RoboDK station: RoboDK_VersionFinal.rdk

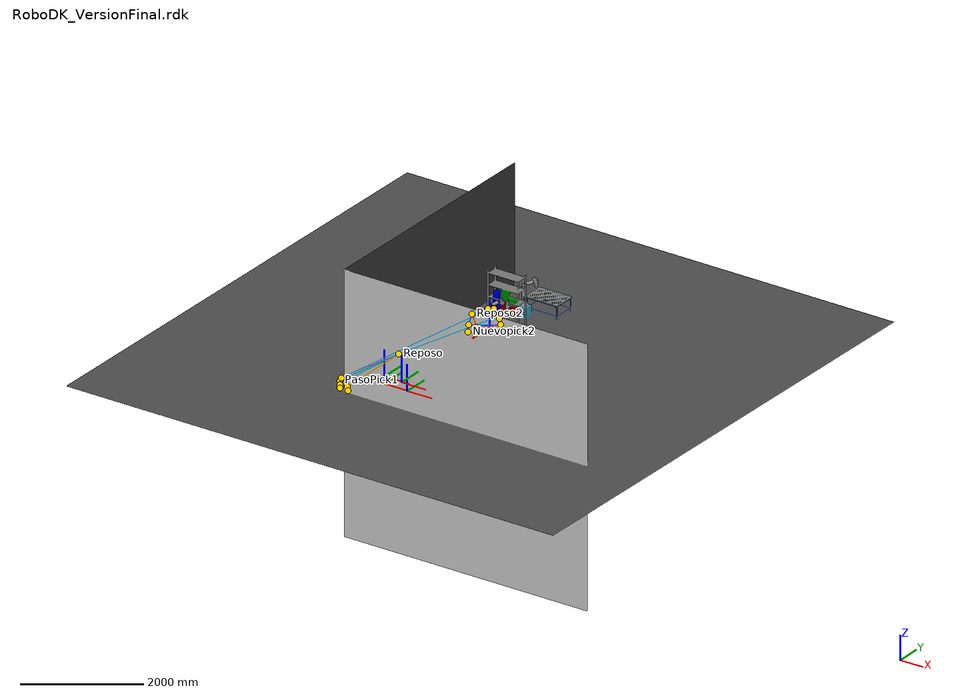
[picture v0: the station drawn from its stored meshes, robots at their saved joint values, targets as dots, program paths as lines]
Station RoboDK_VersionFinal (saved by RoboDK 5.9.4). Poses are relative to the parent item; angles as X-Y-Z fixed-axis rotations.
Station parameters (name, value as stored): IO_5, 1, pedido_id, 3, pedido_tipo, enantyum, pedido_posicion, X01-Y03, pedido_resultado, ok
  - frame UR3e Base - Clasificación at (400, 3450, 0) mm, rotated rx 0 ry 0 rz -90 deg
    - robot UR3e - Clasificaci (model UR3e): 6 axes, payload 3 kg, reach 500 mm, repeatability 0.03 mm, weight 11 kg
        modified DH rows (alpha deg, a mm, theta deg, d mm): 0, 0, 0, 151.9; 90, 0, 180, 0; 0, 243.55, 0, 0; 0, 213.2, 0, 131.05; -90, 0, 0, 85.35; 90, 0, 180, 92.1
        joint limits [-360, -360, -360, -360, -360, -360] to [360, 360, 360, 360, 360, 360]; home [0, -90, -90, 0, 90, 0]; saved at [130.788, -87.81, -66.397, -108.453, 84.697, 21.441]
      - tool RobotiQ EPick Vacuum Gripper (1 Cup), TCP at (0, 0, 130) mm, size 75 x 83 x 136.1 mm
    - target Reposo2 (Cartesian target) at (424.11, -46.06, 399.9) mm, rotated rx -137.59 ry 6.02 rz -87.52 deg; joints [13.28, -91.48, -57.54, -78.3, 87.11, 12.01] of UR3e - Clasificaci
    - object base - clasificaci at (0, 0, -100) mm, rotated rx 90 ry 0 rz 0 deg, size 170 x 200 x 170 mm, geometry from olaquease.obj
  - frame UR3e Base - Despaletizado at (50, 1000, 0) mm
    - robot UR3e - Despaletizado (model UR3e): 6 axes, payload 3 kg, reach 500 mm, repeatability 0.03 mm, weight 11 kg
        modified DH rows (alpha deg, a mm, theta deg, d mm): 0, 0, 0, 151.9; 90, 0, 180, 0; 0, 243.55, 0, 0; 0, 213.2, 0, 131.05; -90, 0, 0, 85.35; 90, 0, 180, 92.1
        joint limits [-360, -360, -360, -360, -360, -360] to [360, 360, 360, 360, 360, 360]; home [0, -90, -90, 0, 90, 0]; saved at [15.698, -84.751, -31.553, -98.733, 77.366, 5.023]
      - tool OnRobot VGP20 Vacuum Gripper, TCP at (-36, 0, 106.49) mm, size 268.4 x 184.1 x 103.7 mm
    - target Reposo (Cartesian target) at (336.1, -92.12, 531.02) mm, rotated rx -124.13 ry -3.06 rz -87.54 deg; joints [0.63, -91.59, -31.74, -90.74, 89.8, -3.56] of UR3e - Despaletizado
    - object base - despaletizado at (0, 0, -100) mm, rotated rx 90 ry 0 rz 0 deg, size 170 x 200 x 170 mm, geometry from olaquease.obj
  - frame cinta - despaletizado at (200, 775, 0) mm
    - robot cinta: 1 axes
        modified DH rows (alpha deg, a mm, theta deg, d mm): 0, 0, 0, 0 linear
        base shift (0, 0, 0) mm, rotated rx 0 ry 90 rz 0 deg
        joint limits [425] to [2000]; home [0]; saved at [450]
      - frame Frame 10 at (0, 0, 0) mm
        - frame Frame_Caja at (-250, 200, 0) mm
          - target Pick1 (Cartesian target) at (139.89, -13.23, 94.59) mm, rotated rx -179.32 ry 0 rz -90.91 deg; joints [11.689, -127.545, -60.36, -81.431, 89.852, 12.598] of UR3e - Despaletizado
          - target Pick2 (Cartesian target) at (-5.95, -20.92, 97.87) mm, rotated rx -179.32 ry 0 rz -90.91 deg; joints [15.948, -91.701, -109.286, -68.363, 89.803, 16.857] of UR3e - Despaletizado
          - target PasoPick (Cartesian target) at (-6.64, 14.1, 202.86) mm, rotated rx -179.32 ry 0 rz -90.91 deg; joints [15.815, -88.174, -90.444, -90.732, 89.804, 16.724] of UR3e - Despaletizado
          - target PasoPick1 (Cartesian target) at (-6.72, -20.9, 162.87) mm, rotated rx -179.32 ry 0 rz -90.91 deg; joints [15.992, -88.247, -94.806, -86.296, 89.802, 16.901] of UR3e - Despaletizado
          - target Pick1-abajo (Cartesian target) at (140.66, -13.24, 29.59) mm, rotated rx -179.32 ry 0 rz -90.91 deg; joints [11.667, -132.164, -70.38, -66.792, 89.852, 12.576] of UR3e - Despaletizado
          - target Pick2-abajo (Cartesian target) at (-5.24, -20.93, 37.87) mm, rotated rx -179.32 ry 0 rz -90.91 deg; joints [15.908, -99.569, -119.052, -50.728, 89.803, 16.817] of UR3e - Despaletizado
        - frame Frame_Caja at (-250, 200, 0) mm
          - target Pick1 (Cartesian target) at (139.89, -13.23, 94.59) mm, rotated rx -179.32 ry 0 rz -90.91 deg; joints [11.689, -127.545, -60.36, -81.431, 89.852, 12.598] of UR3e - Despaletizado
          - target Pick2 (Cartesian target) at (-5.95, -20.92, 97.87) mm, rotated rx -179.32 ry 0 rz -90.91 deg; joints [15.948, -91.701, -109.286, -68.363, 89.803, 16.857] of UR3e - Despaletizado
          - target PasoPick (Cartesian target) at (-6.64, 14.1, 202.86) mm, rotated rx -179.32 ry 0 rz -90.91 deg; joints [15.815, -88.174, -90.444, -90.732, 89.804, 16.724] of UR3e - Despaletizado
          - target PasoPick1 (Cartesian target) at (-6.72, -20.9, 162.87) mm, rotated rx -179.32 ry 0 rz -90.91 deg; joints [15.992, -88.247, -94.806, -86.296, 89.802, 16.901] of UR3e - Despaletizado
          - target Pick1-abajo (Cartesian target) at (140.66, -13.24, 29.59) mm, rotated rx -179.32 ry 0 rz -90.91 deg; joints [11.667, -132.164, -70.38, -66.792, 89.852, 12.576] of UR3e - Despaletizado
          - target Pick2-abajo (Cartesian target) at (-5.24, -20.93, 37.87) mm, rotated rx -179.32 ry 0 rz -90.91 deg; joints [15.908, -99.569, -119.052, -50.728, 89.803, 16.817] of UR3e - Despaletizado
        - frame Frame_Caja at (-250, 200, 0) mm
          - target Pick1 (Cartesian target) at (139.89, -13.23, 94.59) mm, rotated rx -179.32 ry 0 rz -90.91 deg; joints [11.689, -127.545, -60.36, -81.431, 89.852, 12.598] of UR3e - Despaletizado
          - target Pick2 (Cartesian target) at (-5.95, -20.92, 97.87) mm, rotated rx -179.32 ry 0 rz -90.91 deg; joints [15.948, -91.701, -109.286, -68.363, 89.803, 16.857] of UR3e - Despaletizado
          - target PasoPick (Cartesian target) at (-6.64, 14.1, 202.86) mm, rotated rx -179.32 ry 0 rz -90.91 deg; joints [15.815, -88.174, -90.444, -90.732, 89.804, 16.724] of UR3e - Despaletizado
          - target PasoPick1 (Cartesian target) at (-6.72, -20.9, 162.87) mm, rotated rx -179.32 ry 0 rz -90.91 deg; joints [15.992, -88.247, -94.806, -86.296, 89.802, 16.901] of UR3e - Despaletizado
          - target Pick1-abajo (Cartesian target) at (140.66, -13.24, 29.59) mm, rotated rx -179.32 ry 0 rz -90.91 deg; joints [11.667, -132.164, -70.38, -66.792, 89.852, 12.576] of UR3e - Despaletizado
          - target Pick2-abajo (Cartesian target) at (-5.24, -20.93, 37.87) mm, rotated rx -179.32 ry 0 rz -90.91 deg; joints [15.908, -99.569, -119.052, -50.728, 89.803, 16.817] of UR3e - Despaletizado
        - frame Frame_Caja at (-250, 200, 0) mm
          - target Pick1 (Cartesian target) at (139.89, -13.23, 94.59) mm, rotated rx -179.32 ry 0 rz -90.91 deg; joints [11.689, -127.545, -60.36, -81.431, 89.852, 12.598] of UR3e - Despaletizado
          - target Pick2 (Cartesian target) at (-5.95, -20.92, 97.87) mm, rotated rx -179.32 ry 0 rz -90.91 deg; joints [15.948, -91.701, -109.286, -68.363, 89.803, 16.857] of UR3e - Despaletizado
          - target PasoPick (Cartesian target) at (-6.64, 14.1, 202.86) mm, rotated rx -179.32 ry 0 rz -90.91 deg; joints [15.815, -88.174, -90.444, -90.732, 89.804, 16.724] of UR3e - Despaletizado
          - target PasoPick1 (Cartesian target) at (-6.72, -20.9, 162.87) mm, rotated rx -179.32 ry 0 rz -90.91 deg; joints [15.992, -88.247, -94.806, -86.296, 89.802, 16.901] of UR3e - Despaletizado
          - target Pick1-abajo (Cartesian target) at (140.66, -13.24, 29.59) mm, rotated rx -179.32 ry 0 rz -90.91 deg; joints [11.667, -132.164, -70.38, -66.792, 89.852, 12.576] of UR3e - Despaletizado
          - target Pick2-abajo (Cartesian target) at (-5.24, -20.93, 37.87) mm, rotated rx -179.32 ry 0 rz -90.91 deg; joints [15.908, -99.569, -119.052, -50.728, 89.803, 16.817] of UR3e - Despaletizado
        - frame Frame_Caja at (-250, 200, 0) mm
          - target Pick1 (Cartesian target) at (139.89, -13.23, 94.59) mm, rotated rx -179.32 ry 0 rz -90.91 deg; joints [11.689, -127.545, -60.36, -81.431, 89.852, 12.598] of UR3e - Despaletizado
          - target Pick2 (Cartesian target) at (-5.95, -20.92, 97.87) mm, rotated rx -179.32 ry 0 rz -90.91 deg; joints [15.948, -91.701, -109.286, -68.363, 89.803, 16.857] of UR3e - Despaletizado
          - target PasoPick (Cartesian target) at (-6.64, 14.1, 202.86) mm, rotated rx -179.32 ry 0 rz -90.91 deg; joints [15.815, -88.174, -90.444, -90.732, 89.804, 16.724] of UR3e - Despaletizado
          - target PasoPick1 (Cartesian target) at (-6.72, -20.9, 162.87) mm, rotated rx -179.32 ry 0 rz -90.91 deg; joints [15.992, -88.247, -94.806, -86.296, 89.802, 16.901] of UR3e - Despaletizado
          - target Pick1-abajo (Cartesian target) at (140.66, -13.24, 29.59) mm, rotated rx -179.32 ry 0 rz -90.91 deg; joints [11.667, -132.164, -70.38, -66.792, 89.852, 12.576] of UR3e - Despaletizado
          - target Pick2-abajo (Cartesian target) at (-5.24, -20.93, 37.87) mm, rotated rx -179.32 ry 0 rz -90.91 deg; joints [15.908, -99.569, -119.052, -50.728, 89.803, 16.817] of UR3e - Despaletizado
        - frame Frame_Caja at (-250, 200, 0) mm
          - target Pick1 (Cartesian target) at (139.89, -13.23, 94.59) mm, rotated rx -179.32 ry 0 rz -90.91 deg; joints [11.689, -127.545, -60.36, -81.431, 89.852, 12.598] of UR3e - Despaletizado
          - target Pick2 (Cartesian target) at (-5.95, -20.92, 97.87) mm, rotated rx -179.32 ry 0 rz -90.91 deg; joints [15.948, -91.701, -109.286, -68.363, 89.803, 16.857] of UR3e - Despaletizado
          - target PasoPick (Cartesian target) at (-6.64, 14.1, 202.86) mm, rotated rx -179.32 ry 0 rz -90.91 deg; joints [15.815, -88.174, -90.444, -90.732, 89.804, 16.724] of UR3e - Despaletizado
          - target PasoPick1 (Cartesian target) at (-6.72, -20.9, 162.87) mm, rotated rx -179.32 ry 0 rz -90.91 deg; joints [15.992, -88.247, -94.806, -86.296, 89.802, 16.901] of UR3e - Despaletizado
          - target Pick1-abajo (Cartesian target) at (140.66, -13.24, 29.59) mm, rotated rx -179.32 ry 0 rz -90.91 deg; joints [11.667, -132.164, -70.38, -66.792, 89.852, 12.576] of UR3e - Despaletizado
          - target Pick2-abajo (Cartesian target) at (-5.24, -20.93, 37.87) mm, rotated rx -179.32 ry 0 rz -90.91 deg; joints [15.908, -99.569, -119.052, -50.728, 89.803, 16.817] of UR3e - Despaletizado
        - frame Frame_Caja at (-250, 200, 0) mm
          - target Pick1 (Cartesian target) at (139.89, -13.23, 94.59) mm, rotated rx -179.32 ry 0 rz -90.91 deg; joints [11.689, -127.545, -60.36, -81.431, 89.852, 12.598] of UR3e - Despaletizado
          - target Pick2 (Cartesian target) at (-5.95, -20.92, 97.87) mm, rotated rx -179.32 ry 0 rz -90.91 deg; joints [15.948, -91.701, -109.286, -68.363, 89.803, 16.857] of UR3e - Despaletizado
          - target PasoPick (Cartesian target) at (-6.64, 14.1, 202.86) mm, rotated rx -179.32 ry 0 rz -90.91 deg; joints [15.815, -88.174, -90.444, -90.732, 89.804, 16.724] of UR3e - Despaletizado
          - target PasoPick1 (Cartesian target) at (-6.72, -20.9, 162.87) mm, rotated rx -179.32 ry 0 rz -90.91 deg; joints [15.992, -88.247, -94.806, -86.296, 89.802, 16.901] of UR3e - Despaletizado
          - target Pick1-abajo (Cartesian target) at (140.66, -13.24, 29.59) mm, rotated rx -179.32 ry 0 rz -90.91 deg; joints [11.667, -132.164, -70.38, -66.792, 89.852, 12.576] of UR3e - Despaletizado
          - target Pick2-abajo (Cartesian target) at (-5.24, -20.93, 37.87) mm, rotated rx -179.32 ry 0 rz -90.91 deg; joints [15.908, -99.569, -119.052, -50.728, 89.803, 16.817] of UR3e - Despaletizado
        - frame Frame_Caja at (-250, 200, 0) mm
          - target Pick1 (Cartesian target) at (139.89, -13.23, 94.59) mm, rotated rx -179.32 ry 0 rz -90.91 deg; joints [11.689, -127.545, -60.36, -81.431, 89.852, 12.598] of UR3e - Despaletizado
          - target Pick2 (Cartesian target) at (-5.95, -20.92, 97.87) mm, rotated rx -179.32 ry 0 rz -90.91 deg; joints [15.948, -91.701, -109.286, -68.363, 89.803, 16.857] of UR3e - Despaletizado
          - target PasoPick (Cartesian target) at (-6.64, 14.1, 202.86) mm, rotated rx -179.32 ry 0 rz -90.91 deg; joints [15.815, -88.174, -90.444, -90.732, 89.804, 16.724] of UR3e - Despaletizado
          - target PasoPick1 (Cartesian target) at (-6.72, -20.9, 162.87) mm, rotated rx -179.32 ry 0 rz -90.91 deg; joints [15.992, -88.247, -94.806, -86.296, 89.802, 16.901] of UR3e - Despaletizado
          - target Pick1-abajo (Cartesian target) at (140.66, -13.24, 29.59) mm, rotated rx -179.32 ry 0 rz -90.91 deg; joints [11.667, -132.164, -70.38, -66.792, 89.852, 12.576] of UR3e - Despaletizado
          - target Pick2-abajo (Cartesian target) at (-5.24, -20.93, 37.87) mm, rotated rx -179.32 ry 0 rz -90.91 deg; joints [15.908, -99.569, -119.052, -50.728, 89.803, 16.817] of UR3e - Despaletizado
        - frame Frame_Caja at (-250, 200, 0) mm
          - target Pick1 (Cartesian target) at (139.89, -13.23, 94.59) mm, rotated rx -179.32 ry 0 rz -90.91 deg; joints [11.689, -127.545, -60.36, -81.431, 89.852, 12.598] of UR3e - Despaletizado
          - target Pick2 (Cartesian target) at (-5.95, -20.92, 97.87) mm, rotated rx -179.32 ry 0 rz -90.91 deg; joints [15.948, -91.701, -109.286, -68.363, 89.803, 16.857] of UR3e - Despaletizado
          - target PasoPick (Cartesian target) at (-6.64, 14.1, 202.86) mm, rotated rx -179.32 ry 0 rz -90.91 deg; joints [15.815, -88.174, -90.444, -90.732, 89.804, 16.724] of UR3e - Despaletizado
          - target PasoPick1 (Cartesian target) at (-6.72, -20.9, 162.87) mm, rotated rx -179.32 ry 0 rz -90.91 deg; joints [15.992, -88.247, -94.806, -86.296, 89.802, 16.901] of UR3e - Despaletizado
          - target Pick1-abajo (Cartesian target) at (140.66, -13.24, 29.59) mm, rotated rx -179.32 ry 0 rz -90.91 deg; joints [11.667, -132.164, -70.38, -66.792, 89.852, 12.576] of UR3e - Despaletizado
          - target Pick2-abajo (Cartesian target) at (-5.24, -20.93, 37.87) mm, rotated rx -179.32 ry 0 rz -90.91 deg; joints [15.908, -99.569, -119.052, -50.728, 89.803, 16.817] of UR3e - Despaletizado
        - frame Frame_Caja at (-250, 200, 0) mm
          - target Pick1 (Cartesian target) at (139.89, -13.23, 94.59) mm, rotated rx -179.32 ry 0 rz -90.91 deg; joints [11.689, -127.545, -60.36, -81.431, 89.852, 12.598] of UR3e - Despaletizado
          - target Pick2 (Cartesian target) at (-5.95, -20.92, 97.87) mm, rotated rx -179.32 ry 0 rz -90.91 deg; joints [15.948, -91.701, -109.286, -68.363, 89.803, 16.857] of UR3e - Despaletizado
          - target PasoPick (Cartesian target) at (-6.64, 14.1, 202.86) mm, rotated rx -179.32 ry 0 rz -90.91 deg; joints [15.815, -88.174, -90.444, -90.732, 89.804, 16.724] of UR3e - Despaletizado
          - target PasoPick1 (Cartesian target) at (-6.72, -20.9, 162.87) mm, rotated rx -179.32 ry 0 rz -90.91 deg; joints [15.992, -88.247, -94.806, -86.296, 89.802, 16.901] of UR3e - Despaletizado
          - target Pick1-abajo (Cartesian target) at (140.66, -13.24, 29.59) mm, rotated rx -179.32 ry 0 rz -90.91 deg; joints [11.667, -132.164, -70.38, -66.792, 89.852, 12.576] of UR3e - Despaletizado
          - target Pick2-abajo (Cartesian target) at (-5.24, -20.93, 37.87) mm, rotated rx -179.32 ry 0 rz -90.91 deg; joints [15.908, -99.569, -119.052, -50.728, 89.803, 16.817] of UR3e - Despaletizado
        - frame Frame_Caja at (-250, 200, 0) mm
          - target Pick1 (Cartesian target) at (139.89, -13.23, 94.59) mm, rotated rx -179.32 ry 0 rz -90.91 deg; joints [11.689, -127.545, -60.36, -81.431, 89.852, 12.598] of UR3e - Despaletizado
          - target Pick2 (Cartesian target) at (-5.95, -20.92, 97.87) mm, rotated rx -179.32 ry 0 rz -90.91 deg; joints [15.948, -91.701, -109.286, -68.363, 89.803, 16.857] of UR3e - Despaletizado
          - target PasoPick (Cartesian target) at (-6.64, 14.1, 202.86) mm, rotated rx -179.32 ry 0 rz -90.91 deg; joints [15.815, -88.174, -90.444, -90.732, 89.804, 16.724] of UR3e - Despaletizado
          - target PasoPick1 (Cartesian target) at (-6.72, -20.9, 162.87) mm, rotated rx -179.32 ry 0 rz -90.91 deg; joints [15.992, -88.247, -94.806, -86.296, 89.802, 16.901] of UR3e - Despaletizado
          - target Pick1-abajo (Cartesian target) at (140.66, -13.24, 29.59) mm, rotated rx -179.32 ry 0 rz -90.91 deg; joints [11.667, -132.164, -70.38, -66.792, 89.852, 12.576] of UR3e - Despaletizado
          - target Pick2-abajo (Cartesian target) at (-5.24, -20.93, 37.87) mm, rotated rx -179.32 ry 0 rz -90.91 deg; joints [15.908, -99.569, -119.052, -50.728, 89.803, 16.817] of UR3e - Despaletizado
        - frame Frame_Caja at (-250, 200, 0) mm
          - target Pick1 (Cartesian target) at (139.89, -13.23, 94.59) mm, rotated rx -179.32 ry 0 rz -90.91 deg; joints [11.689, -127.545, -60.36, -81.431, 89.852, 12.598] of UR3e - Despaletizado
          - target Pick2 (Cartesian target) at (-5.95, -20.92, 97.87) mm, rotated rx -179.32 ry 0 rz -90.91 deg; joints [15.948, -91.701, -109.286, -68.363, 89.803, 16.857] of UR3e - Despaletizado
          - target PasoPick (Cartesian target) at (-6.64, 14.1, 202.86) mm, rotated rx -179.32 ry 0 rz -90.91 deg; joints [15.815, -88.174, -90.444, -90.732, 89.804, 16.724] of UR3e - Despaletizado
          - target PasoPick1 (Cartesian target) at (-6.72, -20.9, 162.87) mm, rotated rx -179.32 ry 0 rz -90.91 deg; joints [15.992, -88.247, -94.806, -86.296, 89.802, 16.901] of UR3e - Despaletizado
          - target Pick1-abajo (Cartesian target) at (140.66, -13.24, 29.59) mm, rotated rx -179.32 ry 0 rz -90.91 deg; joints [11.667, -132.164, -70.38, -66.792, 89.852, 12.576] of UR3e - Despaletizado
          - target Pick2-abajo (Cartesian target) at (-5.24, -20.93, 37.87) mm, rotated rx -179.32 ry 0 rz -90.91 deg; joints [15.908, -99.569, -119.052, -50.728, 89.803, 16.817] of UR3e - Despaletizado
        - frame Frame_Caja at (-250, 200, 0) mm
          - target Pick1 (Cartesian target) at (139.89, -13.23, 94.59) mm, rotated rx -179.32 ry 0 rz -90.91 deg; joints [11.689, -127.545, -60.36, -81.431, 89.852, 12.598] of UR3e - Despaletizado
          - target Pick2 (Cartesian target) at (-5.95, -20.92, 97.87) mm, rotated rx -179.32 ry 0 rz -90.91 deg; joints [15.948, -91.701, -109.286, -68.363, 89.803, 16.857] of UR3e - Despaletizado
          - target PasoPick (Cartesian target) at (-6.64, 14.1, 202.86) mm, rotated rx -179.32 ry 0 rz -90.91 deg; joints [15.815, -88.174, -90.444, -90.732, 89.804, 16.724] of UR3e - Despaletizado
          - target PasoPick1 (Cartesian target) at (-6.72, -20.9, 162.87) mm, rotated rx -179.32 ry 0 rz -90.91 deg; joints [15.992, -88.247, -94.806, -86.296, 89.802, 16.901] of UR3e - Despaletizado
          - target Pick1-abajo (Cartesian target) at (140.66, -13.24, 29.59) mm, rotated rx -179.32 ry 0 rz -90.91 deg; joints [11.667, -132.164, -70.38, -66.792, 89.852, 12.576] of UR3e - Despaletizado
          - target Pick2-abajo (Cartesian target) at (-5.24, -20.93, 37.87) mm, rotated rx -179.32 ry 0 rz -90.91 deg; joints [15.908, -99.569, -119.052, -50.728, 89.803, 16.817] of UR3e - Despaletizado
        - frame Frame_Caja at (-250, 200, 0) mm
          - target Pick1 (Cartesian target) at (139.89, -13.23, 94.59) mm, rotated rx -179.32 ry 0 rz -90.91 deg; joints [11.689, -127.545, -60.36, -81.431, 89.852, 12.598] of UR3e - Despaletizado
          - target Pick2 (Cartesian target) at (-5.95, -20.92, 97.87) mm, rotated rx -179.32 ry 0 rz -90.91 deg; joints [15.948, -91.701, -109.286, -68.363, 89.803, 16.857] of UR3e - Despaletizado
          - target PasoPick (Cartesian target) at (-6.64, 14.1, 202.86) mm, rotated rx -179.32 ry 0 rz -90.91 deg; joints [15.815, -88.174, -90.444, -90.732, 89.804, 16.724] of UR3e - Despaletizado
          - target PasoPick1 (Cartesian target) at (-6.72, -20.9, 162.87) mm, rotated rx -179.32 ry 0 rz -90.91 deg; joints [15.992, -88.247, -94.806, -86.296, 89.802, 16.901] of UR3e - Despaletizado
          - target Pick1-abajo (Cartesian target) at (140.66, -13.24, 29.59) mm, rotated rx -179.32 ry 0 rz -90.91 deg; joints [11.667, -132.164, -70.38, -66.792, 89.852, 12.576] of UR3e - Despaletizado
          - target Pick2-abajo (Cartesian target) at (-5.24, -20.93, 37.87) mm, rotated rx -179.32 ry 0 rz -90.91 deg; joints [15.908, -99.569, -119.052, -50.728, 89.803, 16.817] of UR3e - Despaletizado
        - frame Frame_Caja at (-250, 200, 0) mm
          - target Pick1 (Cartesian target) at (139.89, -13.23, 94.59) mm, rotated rx -179.32 ry 0 rz -90.91 deg; joints [11.689, -127.545, -60.36, -81.431, 89.852, 12.598] of UR3e - Despaletizado
          - target Pick2 (Cartesian target) at (-5.95, -20.92, 97.87) mm, rotated rx -179.32 ry 0 rz -90.91 deg; joints [15.948, -91.701, -109.286, -68.363, 89.803, 16.857] of UR3e - Despaletizado
          - target PasoPick (Cartesian target) at (-6.64, 14.1, 202.86) mm, rotated rx -179.32 ry 0 rz -90.91 deg; joints [15.815, -88.174, -90.444, -90.732, 89.804, 16.724] of UR3e - Despaletizado
          - target PasoPick1 (Cartesian target) at (-6.72, -20.9, 162.87) mm, rotated rx -179.32 ry 0 rz -90.91 deg; joints [15.992, -88.247, -94.806, -86.296, 89.802, 16.901] of UR3e - Despaletizado
          - target Pick1-abajo (Cartesian target) at (140.66, -13.24, 29.59) mm, rotated rx -179.32 ry 0 rz -90.91 deg; joints [11.667, -132.164, -70.38, -66.792, 89.852, 12.576] of UR3e - Despaletizado
          - target Pick2-abajo (Cartesian target) at (-5.24, -20.93, 37.87) mm, rotated rx -179.32 ry 0 rz -90.91 deg; joints [15.908, -99.569, -119.052, -50.728, 89.803, 16.817] of UR3e - Despaletizado
        - frame Frame_Caja at (-250, 200, 0) mm
          - target Pick1 (Cartesian target) at (139.89, -13.23, 94.59) mm, rotated rx -179.32 ry 0 rz -90.91 deg; joints [11.689, -127.545, -60.36, -81.431, 89.852, 12.598] of UR3e - Despaletizado
          - target Pick2 (Cartesian target) at (-5.95, -20.92, 97.87) mm, rotated rx -179.32 ry 0 rz -90.91 deg; joints [15.948, -91.701, -109.286, -68.363, 89.803, 16.857] of UR3e - Despaletizado
          - target PasoPick (Cartesian target) at (-6.64, 14.1, 202.86) mm, rotated rx -179.32 ry 0 rz -90.91 deg; joints [15.815, -88.174, -90.444, -90.732, 89.804, 16.724] of UR3e - Despaletizado
          - target PasoPick1 (Cartesian target) at (-6.72, -20.9, 162.87) mm, rotated rx -179.32 ry 0 rz -90.91 deg; joints [15.992, -88.247, -94.806, -86.296, 89.802, 16.901] of UR3e - Despaletizado
          - target Pick1-abajo (Cartesian target) at (140.66, -13.24, 29.59) mm, rotated rx -179.32 ry 0 rz -90.91 deg; joints [11.667, -132.164, -70.38, -66.792, 89.852, 12.576] of UR3e - Despaletizado
          - target Pick2-abajo (Cartesian target) at (-5.24, -20.93, 37.87) mm, rotated rx -179.32 ry 0 rz -90.91 deg; joints [15.908, -99.569, -119.052, -50.728, 89.803, 16.817] of UR3e - Despaletizado
        - frame Frame_Caja at (-250, 200, 0) mm
          - target Pick1 (Cartesian target) at (139.89, -13.23, 94.59) mm, rotated rx -179.32 ry 0 rz -90.91 deg; joints [11.689, -127.545, -60.36, -81.431, 89.852, 12.598] of UR3e - Despaletizado
          - target Pick2 (Cartesian target) at (-5.95, -20.92, 97.87) mm, rotated rx -179.32 ry 0 rz -90.91 deg; joints [15.948, -91.701, -109.286, -68.363, 89.803, 16.857] of UR3e - Despaletizado
          - target PasoPick (Cartesian target) at (-6.64, 14.1, 202.86) mm, rotated rx -179.32 ry 0 rz -90.91 deg; joints [15.815, -88.174, -90.444, -90.732, 89.804, 16.724] of UR3e - Despaletizado
          - target PasoPick1 (Cartesian target) at (-6.72, -20.9, 162.87) mm, rotated rx -179.32 ry 0 rz -90.91 deg; joints [15.992, -88.247, -94.806, -86.296, 89.802, 16.901] of UR3e - Despaletizado
          - target Pick1-abajo (Cartesian target) at (140.66, -13.24, 29.59) mm, rotated rx -179.32 ry 0 rz -90.91 deg; joints [11.667, -132.164, -70.38, -66.792, 89.852, 12.576] of UR3e - Despaletizado
          - target Pick2-abajo (Cartesian target) at (-5.24, -20.93, 37.87) mm, rotated rx -179.32 ry 0 rz -90.91 deg; joints [15.908, -99.569, -119.052, -50.728, 89.803, 16.817] of UR3e - Despaletizado
        - frame Frame_Caja at (-250, 200, 0) mm
          - target Pick1 (Cartesian target) at (139.89, -13.23, 94.59) mm, rotated rx -179.32 ry 0 rz -90.91 deg; joints [11.689, -127.545, -60.36, -81.431, 89.852, 12.598] of UR3e - Despaletizado
          - target Pick2 (Cartesian target) at (-5.95, -20.92, 97.87) mm, rotated rx -179.32 ry 0 rz -90.91 deg; joints [15.948, -91.701, -109.286, -68.363, 89.803, 16.857] of UR3e - Despaletizado
          - target PasoPick (Cartesian target) at (-6.64, 14.1, 202.86) mm, rotated rx -179.32 ry 0 rz -90.91 deg; joints [15.815, -88.174, -90.444, -90.732, 89.804, 16.724] of UR3e - Despaletizado
          - target PasoPick1 (Cartesian target) at (-6.72, -20.9, 162.87) mm, rotated rx -179.32 ry 0 rz -90.91 deg; joints [15.992, -88.247, -94.806, -86.296, 89.802, 16.901] of UR3e - Despaletizado
          - target Pick1-abajo (Cartesian target) at (140.66, -13.24, 29.59) mm, rotated rx -179.32 ry 0 rz -90.91 deg; joints [11.667, -132.164, -70.38, -66.792, 89.852, 12.576] of UR3e - Despaletizado
          - target Pick2-abajo (Cartesian target) at (-5.24, -20.93, 37.87) mm, rotated rx -179.32 ry 0 rz -90.91 deg; joints [15.908, -99.569, -119.052, -50.728, 89.803, 16.817] of UR3e - Despaletizado
        - frame Frame_Caja at (-250, 200, 0) mm
          - target Pick1 (Cartesian target) at (139.89, -13.23, 94.59) mm, rotated rx -179.32 ry 0 rz -90.91 deg; joints [11.689, -127.545, -60.36, -81.431, 89.852, 12.598] of UR3e - Despaletizado
          - target Pick2 (Cartesian target) at (-5.95, -20.92, 97.87) mm, rotated rx -179.32 ry 0 rz -90.91 deg; joints [15.948, -91.701, -109.286, -68.363, 89.803, 16.857] of UR3e - Despaletizado
          - target PasoPick (Cartesian target) at (-6.64, 14.1, 202.86) mm, rotated rx -179.32 ry 0 rz -90.91 deg; joints [15.815, -88.174, -90.444, -90.732, 89.804, 16.724] of UR3e - Despaletizado
          - target PasoPick1 (Cartesian target) at (-6.72, -20.9, 162.87) mm, rotated rx -179.32 ry 0 rz -90.91 deg; joints [15.992, -88.247, -94.806, -86.296, 89.802, 16.901] of UR3e - Despaletizado
          - target Pick1-abajo (Cartesian target) at (140.66, -13.24, 29.59) mm, rotated rx -179.32 ry 0 rz -90.91 deg; joints [11.667, -132.164, -70.38, -66.792, 89.852, 12.576] of UR3e - Despaletizado
          - target Pick2-abajo (Cartesian target) at (-5.24, -20.93, 37.87) mm, rotated rx -179.32 ry 0 rz -90.91 deg; joints [15.908, -99.569, -119.052, -50.728, 89.803, 16.817] of UR3e - Despaletizado
        - frame Frame_Caja at (-250, 200, 0) mm
          - target Pick1 (Cartesian target) at (139.89, -13.23, 94.59) mm, rotated rx -179.32 ry 0 rz -90.91 deg; joints [11.689, -127.545, -60.36, -81.431, 89.852, 12.598] of UR3e - Despaletizado
          - target Pick2 (Cartesian target) at (-5.95, -20.92, 97.87) mm, rotated rx -179.32 ry 0 rz -90.91 deg; joints [15.948, -91.701, -109.286, -68.363, 89.803, 16.857] of UR3e - Despaletizado
          - target PasoPick (Cartesian target) at (-6.64, 14.1, 202.86) mm, rotated rx -179.32 ry 0 rz -90.91 deg; joints [15.815, -88.174, -90.444, -90.732, 89.804, 16.724] of UR3e - Despaletizado
          - target PasoPick1 (Cartesian target) at (-6.72, -20.9, 162.87) mm, rotated rx -179.32 ry 0 rz -90.91 deg; joints [15.992, -88.247, -94.806, -86.296, 89.802, 16.901] of UR3e - Despaletizado
          - target Pick1-abajo (Cartesian target) at (140.66, -13.24, 29.59) mm, rotated rx -179.32 ry 0 rz -90.91 deg; joints [11.667, -132.164, -70.38, -66.792, 89.852, 12.576] of UR3e - Despaletizado
          - target Pick2-abajo (Cartesian target) at (-5.24, -20.93, 37.87) mm, rotated rx -179.32 ry 0 rz -90.91 deg; joints [15.908, -99.569, -119.052, -50.728, 89.803, 16.817] of UR3e - Despaletizado
        - frame Frame_Caja at (-250, 200, 0) mm
          - target Pick1 (Cartesian target) at (139.89, -13.23, 94.59) mm, rotated rx -179.32 ry 0 rz -90.91 deg; joints [11.689, -127.545, -60.36, -81.431, 89.852, 12.598] of UR3e - Despaletizado
          - target Pick2 (Cartesian target) at (-5.95, -20.92, 97.87) mm, rotated rx -179.32 ry 0 rz -90.91 deg; joints [15.948, -91.701, -109.286, -68.363, 89.803, 16.857] of UR3e - Despaletizado
          - target PasoPick (Cartesian target) at (-6.64, 14.1, 202.86) mm, rotated rx -179.32 ry 0 rz -90.91 deg; joints [15.815, -88.174, -90.444, -90.732, 89.804, 16.724] of UR3e - Despaletizado
          - target PasoPick1 (Cartesian target) at (-6.72, -20.9, 162.87) mm, rotated rx -179.32 ry 0 rz -90.91 deg; joints [15.992, -88.247, -94.806, -86.296, 89.802, 16.901] of UR3e - Despaletizado
          - target Pick1-abajo (Cartesian target) at (140.66, -13.24, 29.59) mm, rotated rx -179.32 ry 0 rz -90.91 deg; joints [11.667, -132.164, -70.38, -66.792, 89.852, 12.576] of UR3e - Despaletizado
          - target Pick2-abajo (Cartesian target) at (-5.24, -20.93, 37.87) mm, rotated rx -179.32 ry 0 rz -90.91 deg; joints [15.908, -99.569, -119.052, -50.728, 89.803, 16.817] of UR3e - Despaletizado
        - frame Frame_Caja at (-250, 200, 0) mm
          - target Pick1 (Cartesian target) at (139.89, -13.23, 94.59) mm, rotated rx -179.32 ry 0 rz -90.91 deg; joints [11.689, -127.545, -60.36, -81.431, 89.852, 12.598] of UR3e - Despaletizado
          - target Pick2 (Cartesian target) at (-5.95, -20.92, 97.87) mm, rotated rx -179.32 ry 0 rz -90.91 deg; joints [15.948, -91.701, -109.286, -68.363, 89.803, 16.857] of UR3e - Despaletizado
          - target PasoPick (Cartesian target) at (-6.64, 14.1, 202.86) mm, rotated rx -179.32 ry 0 rz -90.91 deg; joints [15.815, -88.174, -90.444, -90.732, 89.804, 16.724] of UR3e - Despaletizado
          - target PasoPick1 (Cartesian target) at (-6.72, -20.9, 162.87) mm, rotated rx -179.32 ry 0 rz -90.91 deg; joints [15.992, -88.247, -94.806, -86.296, 89.802, 16.901] of UR3e - Despaletizado
          - target Pick1-abajo (Cartesian target) at (140.66, -13.24, 29.59) mm, rotated rx -179.32 ry 0 rz -90.91 deg; joints [11.667, -132.164, -70.38, -66.792, 89.852, 12.576] of UR3e - Despaletizado
          - target Pick2-abajo (Cartesian target) at (-5.24, -20.93, 37.87) mm, rotated rx -179.32 ry 0 rz -90.91 deg; joints [15.908, -99.569, -119.052, -50.728, 89.803, 16.817] of UR3e - Despaletizado
    - object pata1 at (50, 20, -200) mm, size 50 x 50 x 150 mm, geometry from Cylinder-50x150mm.sld
    - object pata2 at (50, 410, -200) mm, size 50 x 50 x 150 mm, geometry from Cylinder-50x150mm.sld
    - object pata3 at (2000, 25, -200) mm, size 50 x 50 x 150 mm, geometry from Cylinder-50x150mm.sld
    - object pata4 at (2000, 410, -190) mm, size 50 x 50 x 150 mm, geometry from Cylinder-50x150mm.sld
  - frame cinta - clasificación at (175, 3250, 0) mm, rotated rx 0 ry 0 rz -90 deg
    - robot cinta 2: 1 axes
        modified DH rows (alpha deg, a mm, theta deg, d mm): 0, 0, 0, 0 linear
        base shift (0, 0, 0) mm, rotated rx 0 ry 90 rz 0 deg
        joint limits [-400] to [2000]; home [0]; saved at [-400]
      - frame Frame_despaletizadas at (0, 5050, 0) mm
        - frame Frame_place_desp1 at (0, 150, 0) mm
          - target Paso1 (Cartesian target) at (-13.08, -5145.35, 202.9) mm, rotated rx -179.31 ry 0 rz 56.73 deg; joints [80.175, -87.842, -84.404, -97.123, 89.724, 23.445] of UR3e - Despaletizado
          - target Paso2 (Cartesian target) at (-60.46, -5061.67, 204.51) mm, rotated rx -178.44 ry -3.78 rz 86.72 deg; joints [70.316, -108.237, -61.222, -97.975, 86.819, -16.522] of UR3e - Despaletizado
          - target Place Despaletizado (Cartesian target) at (-95.9, -4983.44, 30.92) mm, rotated rx -178.44 ry 1.22 rz 86.85 deg; joints [60.153, -137.173, -60.813, -71.172, 91.79, -26.668] of UR3e - Despaletizado
          - target PrePlace_despaletizado (Cartesian target) at (-94.48, -4982.44, 81.11) mm, rotated rx -178.44 ry 1.22 rz 86.85 deg; joints [59.961, -134.066, -52.685, -82.412, 91.793, -26.861] of UR3e - Despaletizado
        - frame Frame_place_desp2 at (220, 150, 0) mm
          - target Paso1 (Cartesian target) at (-13.08, -5145.35, 202.9) mm, rotated rx -179.31 ry 0 rz 56.73 deg; joints [80.175, -87.842, -84.404, -97.123, 89.724, 23.445] of UR3e - Despaletizado
          - target Paso2 (Cartesian target) at (-60.46, -5061.67, 204.51) mm, rotated rx -178.44 ry -3.78 rz 86.72 deg; joints [70.316, -108.237, -61.222, -97.975, 86.819, -16.522] of UR3e - Despaletizado
          - target Place Despaletizado (Cartesian target) at (-95.9, -4983.44, 30.92) mm, rotated rx -178.44 ry 1.22 rz 86.85 deg; joints [60.153, -137.173, -60.813, -71.172, 91.79, -26.668] of UR3e - Despaletizado
          - target PrePlace_despaletizado (Cartesian target) at (-94.48, -4982.44, 81.11) mm, rotated rx -178.44 ry 1.22 rz 86.85 deg; joints [59.961, -134.066, -52.685, -82.412, 91.793, -26.861] of UR3e - Despaletizado
        - frame Frame_place_desp3 at (450, 150, 0) mm
          - target Paso1 (Cartesian target) at (-13.08, -5145.35, 202.9) mm, rotated rx -179.31 ry 0 rz 56.73 deg; joints [80.175, -87.842, -84.404, -97.123, 89.724, 23.445] of UR3e - Despaletizado
          - target Paso2 (Cartesian target) at (-60.46, -5061.67, 204.51) mm, rotated rx -178.44 ry -3.78 rz 86.72 deg; joints [70.316, -108.237, -61.222, -97.975, 86.819, -16.522] of UR3e - Despaletizado
          - target Place Despaletizado (Cartesian target) at (-95.9, -4983.44, 30.92) mm, rotated rx -178.44 ry 1.22 rz 86.85 deg; joints [60.153, -137.173, -60.813, -71.172, 91.79, -26.668] of UR3e - Despaletizado
          - target PrePlace_despaletizado (Cartesian target) at (-94.48, -4982.44, 81.11) mm, rotated rx -178.44 ry 1.22 rz 86.85 deg; joints [59.961, -134.066, -52.685, -82.412, 91.793, -26.861] of UR3e - Despaletizado
        - frame Frame_place_desp4 at (650, 150, 0) mm
          - target Paso1 (Cartesian target) at (-13.08, -5145.35, 202.9) mm, rotated rx -179.31 ry 0 rz 56.73 deg; joints [80.175, -87.842, -84.404, -97.123, 89.724, 23.445] of UR3e - Despaletizado
          - target Paso2 (Cartesian target) at (-60.46, -5061.67, 204.51) mm, rotated rx -178.44 ry -3.78 rz 86.72 deg; joints [70.316, -108.237, -61.222, -97.975, 86.819, -16.522] of UR3e - Despaletizado
          - target Place Despaletizado (Cartesian target) at (-95.9, -4983.44, 30.92) mm, rotated rx -178.44 ry 1.22 rz 86.85 deg; joints [60.153, -137.173, -60.813, -71.172, 91.79, -26.668] of UR3e - Despaletizado
          - target PrePlace_despaletizado (Cartesian target) at (-94.48, -4982.44, 81.11) mm, rotated rx -178.44 ry 1.22 rz 86.85 deg; joints [59.961, -134.066, -52.685, -82.412, 91.793, -26.861] of UR3e - Despaletizado
    - object pata1 - 2 at (50, 20, -200) mm, rotated rx 0 ry 0 rz 90 deg, size 50 x 50 x 150 mm, geometry from Cylinder-50x150mm.sld
    - object pata2 - 2 at (50, 410, -200) mm, size 50 x 50 x 150 mm, geometry from Cylinder-50x150mm.sld
    - object pata3 - 2 at (2000, 25, -200) mm, size 50 x 50 x 150 mm, geometry from Cylinder-50x150mm.sld
    - object pata4 - 2 at (2000, 410, -190) mm, size 50 x 50 x 150 mm, geometry from Cylinder-50x150mm.sld
    - frame Frame Pick Clasificacion at (0, 5200, 0) mm
      - target PrePick_clasif2 (Cartesian target) at (232.44, -5084.56, 187.8) mm, rotated rx -179.98 ry -2.95 rz -81.23 deg; joints [4.402, -122.109, -44.04, -103.606, 87.063, -4.376] of UR3e - Clasificaci
      - target Pick_clasif2 (Cartesian target) at (233.47, -5090.86, 62.97) mm, rotated rx -179.46 ry -2.89 rz -91.48 deg; joints [3.54, -124.29, -74.53, -70.89, 87.07, 5] of UR3e - Clasificaci
      - target Pick_clasif1 (Cartesian target) at (232.87, -4940.49, 61.49) mm, rotated rx -179.31 ry -2.87 rz -91.32 deg; joints [23.68, -121.62, -79.01, -69.96, 87.11, 25] of UR3e - Clasificaci
      - target PrePick_clasif1 (Cartesian target) at (231.51, -4934.23, 186.29) mm, rotated rx -179.99 ry -2.95 rz -78.08 deg; joints [24.552, -118.971, -49.099, -102.568, 87.119, 12.649] of UR3e - Clasificaci
      - target Paso (Cartesian target) at (39.67, -4578.8, 252) mm, rotated rx -168.07 ry -0.24 rz -26.24 deg; joints [76.72, -118.97, -36.89, -102.56, 87.11, 12.64] of UR3e - Clasificaci
      - target Paso2 (Cartesian target) at (-348.42, -4656.59, 306.9) mm, rotated rx -173.21 ry -2.13 rz 42.51 deg; joints [138.85, -99.16, -44.86, -119.46, 87.15, 6.05] of UR3e - Clasificaci
      - target Paso4 (Cartesian target) at (-233.56, -4760.65, 389.01) mm, rotated rx -142.29 ry 2.04 rz 42.48 deg; joints [140, -49.13, -75.05, -108.16, 87.01, 7.2] of UR3e - Clasificaci
      - object infrared sensor - proximity sensor (1) at (190, -5250, 0) mm, rotated rx 0 ry 0 rz 90 deg, size 100 x 42.7 x 42.7 mm, geometry from infrared sensor - proximity sensor (1).stl
      - target Nuevopick1 (Cartesian target) at (239.54, -4940.77, 61.55) mm, rotated rx -179.39 ry -1.29 rz -92.71 deg; joints [22.499, -123.163, -76.629, -70.206, 88.576, 25.201] of UR3e - Clasificaci
      - target Nuevopick2 (Cartesian target) at (233.61, -5087.33, 62.84) mm, rotated rx -179.41 ry -1.33 rz -92.4 deg; joints [3.204, -124.422, -74.353, -70.766, 88.621, 5.588] of UR3e - Clasificaci
  - frame Sistema - Estantería at (400, 4050, -173.38) mm
    - target Place 1 (Cartesian target) at (-22.93, -204.87, 525.14) mm, rotated rx -90 ry 0 rz 0 deg; joints [207.93, -116.903, -92.388, 29.291, 62.07, 0] of UR3e - Clasificaci
    - target Target 2 (Cartesian target) at (322.8, -521.68, 452.98) mm, rotated rx -171.23 ry -2.21 rz -71.16 deg; joints [130.788, -87.631, -67.051, -107.978, 84.697, 21.441] of UR3e - Clasificaci
    - target Place_base (Cartesian target) at (-213.83, -204.87, 379.68) mm, rotated rx -90 ry 0 rz 0 deg; joints [259.472, -135.813, -115.812, 71.625, 10.528, 0] of UR3e - Clasificaci
    - object Estanteria at (0, 0, 0) mm, size 624.2 x 963.2 x 234 mm, geometry from eb_metal_shelf_01.obj
    - target Target 3 (Cartesian target) at (400.79, -632.87, 393.4) mm, rotated rx -168.07 ry -0.24 rz -116.24 deg; joints [109.466, -99.497, -72.038, -90.245, 81.324, 45.055] of UR3e - Clasificaci
    - target Pick_base_antes (Cartesian target) at (-213.89, -129.51, 378.2) mm, rotated rx -89.91 ry 1.64 rz 177.07 deg; joints [-103.271, -145.254, -88.344, 53.694, 100.334, 1.652] of UR3e - pedidos
    - target Paso_ped3 (Cartesian target) at (-131.82, 121.32, 662.13) mm, rotated rx -90.23 ry 1.63 rz -178.38 deg; joints [-98.637, -52.41, -111.868, -15.952, 100.265, 1.587] of UR3e - pedidos
    - target Paso_ped4 (Cartesian target) at (-126.77, 42.59, 563.07) mm, rotated rx -90.23 ry 1.63 rz -178.38 deg; joints [-91.201, -64.707, -134.036, 18.516, 92.829, 1.617] of UR3e - pedidos
    - target Paso_ped5 (Cartesian target) at (-214.08, 164.54, 606.19) mm, rotated rx -90.23 ry 1.63 rz -178.38 deg; joints [-135.362, -83.287, -109.019, 11.974, 136.989, 1.385] of UR3e - pedidos
    - target Paso_ped6 (Cartesian target) at (-291.93, 214.82, 509.51) mm, rotated rx -90.23 ry 1.63 rz -178.38 deg; joints [-161.185, -113.423, -102.583, 35.24, 162.811, 0.896] of UR3e - pedidos
    - target Pick_base (Cartesian target) at (-192.17, -40.89, 371.84) mm, rotated rx -88.66 ry 1.64 rz 177.07 deg; joints [18.618, -41.504, 115.771, 102.085, 338.369, -354.973] of UR3e - pedidos
    - object Prism 9-2 at (-148.31, -139.79, 308.56) mm, rotated rx 17.47 ry 88.43 rz -72.45 deg, size 62.5 x 125 x 62.5 mm, geometry from Prism-250x125x125mm.sld
    - object Prism 10-2 at (-0.05, -141.61, 308.76) mm, rotated rx 6.04 ry 88.51 rz -83.84 deg, size 62.5 x 125 x 62.5 mm, geometry from Prism-250x125x125mm.sld
    - object Prism 7-2 at (164.42, -138.64, 308.62) mm, rotated rx 17.47 ry 88.43 rz -72.45 deg, size 62.5 x 125 x 62.5 mm, geometry from Prism-250x125x125mm.sld
    - object Prism 8-2 at (-152.32, -140.45, 523.8) mm, rotated rx 6.04 ry 88.51 rz -83.84 deg, size 62.5 x 125 x 62.5 mm, geometry from Prism-250x125x125mm.sld
    - object Prism 5-2 at (12.15, -137.48, 523.67) mm, rotated rx 17.47 ry 88.43 rz -72.45 deg, size 62.5 x 125 x 62.5 mm, geometry from Prism-250x125x125mm.sld
    - object Prism 6-2 at (160.41, -139.29, 523.84) mm, rotated rx 6.04 ry 88.51 rz -83.84 deg, size 62.5 x 125 x 62.5 mm, geometry from Prism-250x125x125mm.sld
    - object Prism 3-2 at (-137.85, -135.49, 368.76) mm, rotated rx 17.47 ry 88.43 rz -72.45 deg, size 62.5 x 125 x 62.5 mm, geometry from Prism-250x125x125mm.sld
    - object Prism 4-2 at (10.37, -137.3, 368.89) mm, rotated rx 6.04 ry 88.51 rz -83.84 deg, size 62.5 x 125 x 62.5 mm, geometry from Prism-250x125x125mm.sld
    - object Prism 1-2 at (174.88, -134.33, 368.81) mm, rotated rx 17.47 ry 88.43 rz -72.45 deg, size 62.5 x 125 x 62.5 mm, geometry from Prism-250x125x125mm.sld
    - object Prism 2-2 at (-141.9, -136.14, 583.93) mm, rotated rx 6.04 ry 88.51 rz -83.84 deg, size 62.5 x 125 x 62.5 mm, geometry from Prism-250x125x125mm.sld
    - object Prism 9 at (7.18, -144.86, 580.48) mm, rotated rx 17.47 ry 88.43 rz -72.45 deg, size 62.5 x 125 x 62.5 mm, geometry from Prism-250x125x125mm.sld
    - object Prism 7 at (-145.09, -143.7, 431.53) mm, rotated rx 17.47 ry 88.43 rz -72.45 deg, size 62.5 x 125 x 62.5 mm, geometry from Prism-250x125x125mm.sld
    - object Prism 8 at (3.12, -145.52, 431.71) mm, rotated rx 6.04 ry 88.51 rz -83.84 deg, size 62.5 x 125 x 62.5 mm, geometry from Prism-250x125x125mm.sld
    - object Prism 3 at (17.16, -135.47, 643.47) mm, rotated rx 17.47 ry 88.43 rz -72.45 deg, size 62.5 x 125 x 62.5 mm, geometry from Prism-250x125x125mm.sld
  - frame Frame 6 at (-250, 200, 0) mm
    - object tinker at (0, 0, -10) mm, size 400 x 300 x 125 mm, geometry from tinker.obj
    - target Pick1 (Cartesian target) at (139.89, -13.23, 94.59) mm, rotated rx -179.32 ry 0 rz -90.91 deg; joints [11.689, -127.545, -60.36, -81.431, 89.852, 12.598] of UR3e - Despaletizado
    - target Pick2 (Cartesian target) at (-5.95, -20.92, 97.87) mm, rotated rx -179.32 ry 0 rz -90.91 deg; joints [15.948, -91.701, -109.286, -68.363, 89.803, 16.857] of UR3e - Despaletizado
    - target PasoPick (Cartesian target) at (-6.64, 14.1, 202.86) mm, rotated rx -179.32 ry 0 rz -90.91 deg; joints [15.815, -88.174, -90.444, -90.732, 89.804, 16.724] of UR3e - Despaletizado
    - target PasoPick1 (Cartesian target) at (-6.72, -20.9, 162.87) mm, rotated rx -179.32 ry 0 rz -90.91 deg; joints [15.992, -88.247, -94.806, -86.296, 89.802, 16.901] of UR3e - Despaletizado
    - target Pick1-abajo (Cartesian target) at (140.66, -13.24, 29.59) mm, rotated rx -179.32 ry 0 rz -90.91 deg; joints [11.667, -132.164, -70.38, -66.792, 89.852, 12.576] of UR3e - Despaletizado
    - target Pick2-abajo (Cartesian target) at (-5.24, -20.93, 37.87) mm, rotated rx -179.32 ry 0 rz -90.91 deg; joints [15.908, -99.569, -119.052, -50.728, 89.803, 16.817] of UR3e - Despaletizado
    - object Prism 2-2 at (-80, 90, 60) mm, size 62.5 x 125 x 62.5 mm, geometry from Prism-250x125x125mm.sld
    - object Prism 1-2 at (-80, -50, 60) mm, size 62.5 x 125 x 62.5 mm, geometry from Prism-250x125x125mm.sld
    - object Prism 4-2 at (-10, 90, 60) mm, size 62.5 x 125 x 62.5 mm, geometry from Prism-250x125x125mm.sld
    - object Prism 3-2 at (-10, -50, 60) mm, size 62.5 x 125 x 62.5 mm, geometry from Prism-250x125x125mm.sld
    - object Prism 5-2 at (60, -50, 60) mm, size 62.5 x 125 x 62.5 mm, geometry from Prism-250x125x125mm.sld
    - object Prism 6-2 at (60, 90, 60) mm, size 62.5 x 125 x 62.5 mm, geometry from Prism-250x125x125mm.sld
    - object Prism 9-2 at (200, -50, 60) mm, size 62.5 x 125 x 62.5 mm, geometry from Prism-250x125x125mm.sld
    - object Prism 10-2 at (200, 90, 60) mm, size 62.5 x 125 x 62.5 mm, geometry from Prism-250x125x125mm.sld
    - object Prism 7-2 at (130, -50, 60) mm, size 62.5 x 125 x 62.5 mm, geometry from Prism-250x125x125mm.sld
    - object Prism 8-2 at (130, 90, 60) mm, size 62.5 x 125 x 62.5 mm, geometry from Prism-250x125x125mm.sld
    - object Prism 2 at (-80, 90, 0) mm, size 62.5 x 125 x 62.5 mm, geometry from Prism-250x125x125mm.sld
    - object Prism 250x125x125mm at (-80, -50, 0) mm, size 62.5 x 125 x 62.5 mm, geometry from Prism-250x125x125mm.sld
    - object Prism 4 at (-10, 90, 0) mm, size 62.5 x 125 x 62.5 mm, geometry from Prism-250x125x125mm.sld
    - object Prism 3 at (-10, -50, 0) mm, size 62.5 x 125 x 62.5 mm, geometry from Prism-250x125x125mm.sld
    - object Prism 5 at (60, -50, 0) mm, size 62.5 x 125 x 62.5 mm, geometry from Prism-250x125x125mm.sld
    - object Prism 6 at (60, 90, 0) mm, size 62.5 x 125 x 62.5 mm, geometry from Prism-250x125x125mm.sld
    - object Prism 9 at (200, -50, 0) mm, size 62.5 x 125 x 62.5 mm, geometry from Prism-250x125x125mm.sld
    - object Prism 10 at (200, 90, 0) mm, size 62.5 x 125 x 62.5 mm, geometry from Prism-250x125x125mm.sld
    - object Prism 7 at (130, -50, 0) mm, size 62.5 x 125 x 62.5 mm, geometry from Prism-250x125x125mm.sld
    - object Prism 8 at (130, 90, 0) mm, size 62.5 x 125 x 62.5 mm, geometry from Prism-250x125x125mm.sld
  - frame Frame_sensor at (-50, 500, 0) mm
    - object infrared sensor - proximity sensor (1) at (300, 200, 0) mm, rotated rx 0 ry 0 rz 90 deg, size 100 x 42.7 x 42.7 mm, geometry from infrared sensor - proximity sensor (1).stl
  - frame UR3e Base - pedidos at (400, 4430, 0) mm
    - robot UR3e - pedidos (model UR3e): 6 axes, payload 3 kg, reach 500 mm, repeatability 0.03 mm, weight 11 kg
        modified DH rows (alpha deg, a mm, theta deg, d mm): 0, 0, 0, 151.9; 90, 0, 180, 0; 0, 243.55, 0, 0; 0, 213.2, 0, 131.05; -90, 0, 0, 85.35; 90, 0, 180, 92.1
        joint limits [-360, -360, -360, -360, -360, -360] to [360, 360, 360, 360, 360, 360]; home [0, -90, -90, 0, 90, 0]; saved at [33.678, -87.094, -74.931, 0.727, 9.729, -13.917]
      - tool RobotiQ EPick Vacuum Gripper (1 Cup), TCP at (0, 0, 130) mm, size 75 x 83 x 136.1 mm
    - object base - pedidos at (0, 0, -100) mm, rotated rx 90 ry 0 rz 0 deg, size 170 x 200 x 170 mm, geometry from olaquease.obj
    - object Mesa_pedidos at (0, 400, 65) mm, size 636.3 x 422.1 x 252 mm, geometry from Table-2000x1200x800mm.sld
    - frame Frame_pedidos at (0, 400, 65) mm
      - target Place_pedido (Cartesian target) at (384.34, -165.38, 46.78) mm, rotated rx -90.39 ry 0.12 rz -1.35 deg; joints [22.113, -167.141, -69.546, 55.718, 156.539, -0.769] of UR3e - pedidos
      - target Pre_pedidos (Cartesian target) at (383.36, -207.27, 47.06) mm, rotated rx -90.39 ry 0.12 rz -1.35 deg; joints [15.783, -167.001, -69.826, 55.518, 162.867, -1.131] of UR3e - pedidos
      - target Paso_ped2 (Cartesian target) at (474.36, -412.99, 243.96) mm, rotated rx -84.74 ry -1.58 rz -64.81 deg; joints [4.98, -121.46, -105.569, 52.639, 110.266, 0.365] of UR3e - pedidos
      - target Paso_ped1 (Cartesian target) at (421, -495.79, 270.65) mm, rotated rx -84.67 ry 1.35 rz -95.59 deg; joints [17.594, -99.316, -130.185, 55.297, 66.796, -0.937] of UR3e - pedidos
      - target Reposo_pedidos (Cartesian target) at (359.35, -581.08, 488.81) mm, rotated rx -86.88 ry 4.53 rz -136.85 deg; joints [33.678, -87.094, -74.931, 0.727, 9.729, -13.917] of UR3e - pedidos
  - folder Clasificacion
    - program Pick2 (14 instructions, listed below)
    - program Pick1 (14 instructions, listed below)
  - folder Despaletizado
    - program PickPlace-Despaletizado1 (39 instructions, listed below)
    - program PickPlace-Despaletizado2 (33 instructions, listed below)
    - program PickPlace-Despaletizado3 (38 instructions, listed below)
    - program PickPlace-Despaletizado4 (34 instructions, listed below)
    - program Programa Despaletizado (22 instructions, listed below)
  - folder Python
    - Python program Reset (listed below)
    - Python program ApareceCaja (listed below)
    - Python program AvanzaCaja (listed below)
    - Python program CintaPick (listed below)
    - Python program AvanzaPlace (listed below)
    - Python program ResetPick (listed below)
    - Python program AvanzaPick (listed below)
    - Python program ProgramaClasificacion (listed below)
    - Python program Pedidos_PickPlace_base (listed below)
    - Python program Pedidos_PickPlace (listed below)
  - program ProgramaPrincipal (2 instructions, listed below)
  - object Square at (600, 2900, -200) mm, size 9600 x 9600 x 0 mm, geometry from Square.sld
    - object Square at (3800, 0, -200) mm, rotated rx 90 ry 0 rz 90 deg, size 4800 x 4800 x 0 mm, geometry from Square.sld
    - object Square at (-1000, 0, -200) mm, rotated rx 0 ry 90 rz 0 deg, size 4800 x 4800 x 0 mm, geometry from Square.sld
    - object Box 400x200mm (Closed) at (1200, -2200, 0) mm, rotated rx 90 ry 0 rz 90 deg, size 603.6 x 1201.8 x 650 mm, geometry from Box-400x200mm-Closed.sld
    - object Square at (1400, 2400, -200) mm, rotated rx 90 ry 0 rz 0 deg, size 4800 x 4800 x 0 mm, geometry from Square.sld
    - object Square at (1400, -2400, -200) mm, rotated rx 90 ry 0 rz 0 deg, size 4800 x 4800 x 0 mm, geometry from Square.sld
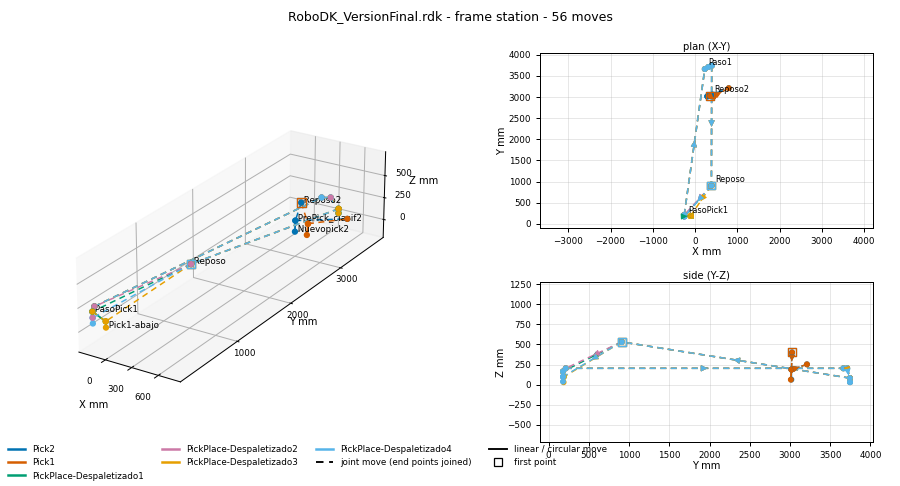
[picture p0: tool path of RoboDK_VersionFinal.rdk in frame station, 56 of 56 moves have a stored position in this frame; points joined in program order, loops and branches not executed]

--- program Pick2 (robot UR3e - Clasificaci) ---
  Est. Ref.: UR3e Base - Clasificación
  Establecer velocidad (500.0 mm/s)
  Est. herr: RobotiQ EPick Vacuum Gripper (1 Cup)
  MoveJ (Reposo2)
  Est. Ref.: Frame Pick Clasificacion
  MoveJ (PrePick_clasif2)
  Establecer velocidad (100.0 mm/s)
  MoveL (Nuevopick2)
  Set IO_5=1
  Adjuntar a RobotiQ EPick Vacuum Gripper (1 Cup)
  Pausa 2.0 s
  MoveL (PrePick_clasif2)
  Establecer velocidad (500.0 mm/s)
  MoveJ (Paso)

--- program Pick1 (robot UR3e - Clasificaci) ---
  Est. Ref.: UR3e Base - Clasificación
  Establecer velocidad (500.0 mm/s)
  Est. herr: RobotiQ EPick Vacuum Gripper (1 Cup)
  MoveJ (Reposo2)
  Est. Ref.: Frame Pick Clasificacion
  MoveJ (PrePick_clasif1)
  Establecer velocidad (100.0 mm/s)
  MoveL (Nuevopick1)
  Set IO_5=1
  Adjuntar a RobotiQ EPick Vacuum Gripper (1 Cup)
  Pausa 2.0 s
  MoveL (PrePick_clasif1)
  Establecer velocidad (500.0 mm/s)
  MoveJ (Paso)

--- program PickPlace-Despaletizado1 (robot UR3e - Despaletizado) ---
  Est. Ref.: UR3e Base - Despaletizado
  Establecer velocidad (500.0 mm/s)
  Est. herr: RobotiQ EPick Vacuum Gripper (1 Cup)
  MoveJ (Reposo)
  Est. Ref.: Frame_6_Copia at (350, -25, 0) mm
  MoveJ (PasoPick1)
  Establecer velocidad (100.0 mm/s)
  MoveL (Pick1)
  Set IO_5=1
  Adjuntar a OnRobot VGP20 Vacuum Gripper
  Adjuntar a OnRobot VGP20 Vacuum Gripper
  Adjuntar a OnRobot VGP20 Vacuum Gripper
  Adjuntar a OnRobot VGP20 Vacuum Gripper
  Adjuntar a OnRobot VGP20 Vacuum Gripper
  Adjuntar a OnRobot VGP20 Vacuum Gripper
  Pausa 2.0 s
  MoveL (PasoPick1)
  Establecer velocidad (500.0 mm/s)
  MoveJ (PasoPick)
  Est. Ref.: Frame_place_desp -> Frame_place_desp1
  MoveJ (Paso1)
  MoveJ (Paso2)
  MoveJ (PrePlace_despaletizado)
  Establecer velocidad (100.0 mm/s)
  MoveL (Place Despaletizado)
  Set IO_5=0
  Est. Ref.: Frame_despaletizadas
  Separar de OnRobot VGP20 Vacuum Gripper
  Separar de OnRobot VGP20 Vacuum Gripper
  Separar de OnRobot VGP20 Vacuum Gripper
  Separar de OnRobot VGP20 Vacuum Gripper
  Separar de OnRobot VGP20 Vacuum Gripper
  Separar de OnRobot VGP20 Vacuum Gripper
  Pausa 2.0 s
  Est. Ref.: Frame_place_desp -> Frame_place_desp1
  MoveL (PrePlace_despaletizado)
  Establecer velocidad (500.0 mm/s)
  Est. Ref.: UR3e Base - Despaletizado
  MoveJ (Reposo)

--- program PickPlace-Despaletizado2 (robot UR3e - Despaletizado) ---
  Est. Ref.: UR3e Base - Despaletizado
  Establecer velocidad (500.0 mm/s)
  Est. herr: RobotiQ EPick Vacuum Gripper (1 Cup)
  MoveJ (Reposo)
  Est. Ref.: Frame_6_Copia at (350, -25, 0) mm
  MoveJ (PasoPick)
  Establecer velocidad (100.0 mm/s)
  MoveL (Pick2)
  Set IO_5=1
  Adjuntar a OnRobot VGP20 Vacuum Gripper
  Adjuntar a OnRobot VGP20 Vacuum Gripper
  Adjuntar a OnRobot VGP20 Vacuum Gripper
  Adjuntar a OnRobot VGP20 Vacuum Gripper
  Pausa 2.0 s
  MoveL (PasoPick1)
  Establecer velocidad (500.0 mm/s)
  MoveJ (PasoPick)
  Est. Ref.: Frame_place_desp2
  MoveJ (Paso1)
  MoveJ (Paso2)
  MoveJ (PrePlace_despaletizado)
  Establecer velocidad (100.0 mm/s)
  MoveL (Place Despaletizado)
  Set IO_5=0
  Separar de OnRobot VGP20 Vacuum Gripper
  Separar de OnRobot VGP20 Vacuum Gripper
  Separar de OnRobot VGP20 Vacuum Gripper
  Separar de OnRobot VGP20 Vacuum Gripper
  Pausa 2.0 s
  MoveL (PrePlace_despaletizado)
  Establecer velocidad (500.0 mm/s)
  Est. Ref.: UR3e Base - Despaletizado
  MoveJ (Reposo)

--- program PickPlace-Despaletizado3 (robot UR3e - Despaletizado) ---
  Est. Ref.: UR3e Base - Despaletizado
  Establecer velocidad (500.0 mm/s)
  Est. herr: RobotiQ EPick Vacuum Gripper (1 Cup)
  MoveJ (Reposo)
  Est. Ref.: Frame_6_Copia at (350, -25, 0) mm
  MoveJ (Pick1)
  Establecer velocidad (100.0 mm/s)
  MoveL (Pick1-abajo)
  Set IO_5=1
  Adjuntar a OnRobot VGP20 Vacuum Gripper
  Adjuntar a OnRobot VGP20 Vacuum Gripper
  Adjuntar a OnRobot VGP20 Vacuum Gripper
  Adjuntar a OnRobot VGP20 Vacuum Gripper
  Adjuntar a OnRobot VGP20 Vacuum Gripper
  Adjuntar a OnRobot VGP20 Vacuum Gripper
  Pausa 2.0 s
  MoveL (Pick1)
  Establecer velocidad (500.0 mm/s)
  MoveJ (PasoPick1)
  MoveJ (PasoPick)
  Est. Ref.: Frame_place_desp3
  MoveJ (Paso1)
  MoveJ (Paso2)
  MoveJ (PrePlace_despaletizado)
  Establecer velocidad (100.0 mm/s)
  MoveL (Place Despaletizado)
  Set IO_5=0
  Separar de OnRobot VGP20 Vacuum Gripper
  Separar de OnRobot VGP20 Vacuum Gripper
  Separar de OnRobot VGP20 Vacuum Gripper
  Separar de OnRobot VGP20 Vacuum Gripper
  Separar de OnRobot VGP20 Vacuum Gripper
  Separar de OnRobot VGP20 Vacuum Gripper
  Pausa 2.0 s
  MoveL (PrePlace_despaletizado)
  Establecer velocidad (500.0 mm/s)
  Est. Ref.: UR3e Base - Despaletizado
  MoveJ (Reposo)

--- program PickPlace-Despaletizado4 (robot UR3e - Despaletizado) ---
  Est. Ref.: UR3e Base - Despaletizado
  Establecer velocidad (500.0 mm/s)
  Est. herr: RobotiQ EPick Vacuum Gripper (1 Cup)
  MoveJ (Reposo)
  Est. Ref.: Frame_6_Copia at (350, -25, 0) mm
  MoveJ (Pick2)
  Establecer velocidad (100.0 mm/s)
  MoveL (Pick2-abajo)
  Set IO_5=1
  Adjuntar a OnRobot VGP20 Vacuum Gripper
  Adjuntar a OnRobot VGP20 Vacuum Gripper
  Adjuntar a OnRobot VGP20 Vacuum Gripper
  Adjuntar a OnRobot VGP20 Vacuum Gripper
  Pausa 2.0 s
  MoveL (Pick2)
  Establecer velocidad (500.0 mm/s)
  MoveJ (PasoPick1)
  MoveJ (PasoPick)
  Est. Ref.: Frame_place_desp4
  MoveJ (Paso1)
  MoveJ (Paso2)
  MoveJ (Place Despaletizado)
  Establecer velocidad (100.0 mm/s)
  MoveL (Place Despaletizado)
  Set IO_5=0
  Separar de OnRobot VGP20 Vacuum Gripper
  Separar de OnRobot VGP20 Vacuum Gripper
  Separar de OnRobot VGP20 Vacuum Gripper
  Pausa 2.0 s
  Separar de OnRobot VGP20 Vacuum Gripper
  MoveL (PrePlace_despaletizado)
  Establecer velocidad (500.0 mm/s)
  Est. Ref.: UR3e Base - Despaletizado
  MoveJ (Reposo)

--- program Programa Despaletizado (robot cinta) ---
  Llamar Reset
  Llamar ResetPick
  Llamar ApareceCaja
  Llamar AvanzaCaja
  Llamar PickPlace-Despaletizado1
  Llamar AvanzaPlace
  Llamar AvanzaPlace
  Llamar AvanzaPlace
  Llamar AvanzaPlace
  Llamar AvanzaPlace
  Llamar PickPlace-Despaletizado2
  Llamar AvanzaPlace
  Llamar AvanzaPlace
  Llamar AvanzaPlace
  Llamar AvanzaPlace
  Llamar PickPlace-Despaletizado3
  Llamar AvanzaPlace
  Llamar AvanzaPlace
  Llamar AvanzaPlace
  Llamar AvanzaPlace
  Llamar PickPlace-Despaletizado4
  Llamar CintaPick

--- Python program Reset ---
# Type help("robodk.robolink") or help("robodk.robomath") for more information
# Press F5 to run the script
# Documentation: https://robodk.com/doc/en/RoboDK-API.html
# Reference:     https://robodk.com/doc/en/PythonAPI/robodk.html
# Note: It is not required to keep a copy of this file, your Python script is saved with your RDK project

# You can also use the new version of the API:
from robodk import robolink    # RoboDK API
from robodk import robomath    # Robot toolbox
RDK = robolink.Robolink()

cinta = RDK.Item('cinta')

if cinta.Valid():
    cinta.setJoints([2000])

--- Python program ApareceCaja ---
# Type help("robodk.robolink") or help("robodk.robomath") for more information
# Press F5 to run the script
# Documentation: https://robodk.com/doc/en/RoboDK-API.html
# Reference:     https://robodk.com/doc/en/PythonAPI/robodk.html

from robodk import robolink    # RoboDK API
from robodk import robomath    # Robot toolbox

RDK = robolink.Robolink()

cinta = RDK.Item('cinta')
INCREMENTO_MM = -1550
caja_grande = RDK.Item('tinker')
caja_grande.setParam('Collisions', '0')


# Conjunto original (Frame con TODAS las cajitas + tinker)
caja = RDK.Item('Frame 6')
tinker = RDK.Item('Frame_6_Copia')

# Frame de la cinta
SR_Cinta = RDK.Item('Frame 10')

def hacer_visible_recursivo(item):

    # Si es un target -> ocultarlo
    if item.Type() == robolink.ITEM_TYPE_TARGET:
        item.setVisible(False)
    else:
        item.setVisible(True)

    # Recorrer hijos
    for hijo in item.Childs():
        hacer_visible_recursivo(hijo)

if cinta.Valid() and caja.Valid():
    # -------------------------------------------------
    # BORRAR COPIAS EXISTENTES EN "Sistema - Estantería"
    # -------------------------------------------------
    estanteria = RDK.Item('Sistema - Estantería')

    if estanteria.Valid():
        hijos = estanteria.Childs()  # copia de la lista
        for item in hijos:
            if item.Valid() and item.Name().startswith('Prism'):
                item.Delete()

    if tinker.Valid():
        tinker.Delete()

    #Copiar una caja
    caja.Copy()
    caja_copia = RDK.Paste()
    caja_copia.setName('Frame_Caja')

    # Colocar la copia en el inicio de la cinta
    caja_copia.setParent(SR_Cinta)
    caja_copia.setPose(caja.Pose())
    caja_copia.setVisible(True)

    hacer_visible_recursivo(caja_copia)

--- Python program AvanzaCaja ---
# Type help("robodk.robolink") or help("robodk.robomath") for more information
# Press F5 to run the script
# Documentation: https://robodk.com/doc/en/RoboDK-API.html
# Reference:     https://robodk.com/doc/en/PythonAPI/robodk.html
# Note: It is not required to keep a copy of this file, your Python script is saved with your RDK project

# You can also use the new version of the API:
from robodk import robolink    # RoboDK API
from robodk import robomath    # Robot toolbox
RDK = robolink.Robolink()

cinta = RDK.Item('cinta')
INCREMENTO_MM = -1550
caja_grande = RDK.Item('tinker')
caja_grande.setParam('Collisions', '0')


# Conjunto original (Frame con TODAS las cajitas + tinker)
caja = RDK.Item('Frame 6')
tinker = RDK.Item('Frame_6_Copia')

if cinta.Valid() and caja.Valid():

    # Avanzar Cinta
    cinta.setSpeed(1000)
    cinta.setAcceleration(100)

    joints = cinta.Joints()
    joints[0] += INCREMENTO_MM
    cinta.MoveJ(joints)

--- Python program CintaPick ---
# Type help("robodk.robolink") or help("robodk.robomath") for more information
# Press F5 to run the script
# Documentation: https://robodk.com/doc/en/RoboDK-API.html
# Reference:     https://robodk.com/doc/en/PythonAPI/robodk.html
# Note: It is not required to keep a copy of this file, your Python script is saved with your RDK project

# You can also use the new version of the API:
from robodk import robolink    # RoboDK API
from robodk import robomath    # Robot toolbox
RDK = robolink.Robolink()

cinta = RDK.Item('cinta 2')
INCREMENTO_MM = -960
#caja = RDK.Item('Frame 11')
SR_Cinta = RDK.Item('Frame_despaletizadas')

if cinta.Valid():
    cinta.setSpeed(500)
    cinta.setAcceleration(500)
    cinta.MoveJ(cinta.Joints() + INCREMENTO_MM)

--- Python program AvanzaPlace ---
# Type help("robodk.robolink") or help("robodk.robomath") for more information
# Press F5 to run the script
# Documentation: https://robodk.com/doc/en/RoboDK-API.html
# Reference:     https://robodk.com/doc/en/PythonAPI/robodk.html
# Note: It is not required to keep a copy of this file, your Python script is saved with your RDK project

# You can also use the new version of the API:
from robodk import robolink    # RoboDK API
from robodk import robomath    # Robot toolbox
RDK = robolink.Robolink()

cinta = RDK.Item('cinta 2')
INCREMENTO_MM = -50
#caja = RDK.Item('Frame 11')
SR_Cinta = RDK.Item('Frame 11')

if cinta.Valid():
    cinta.setSpeed(200)        # velocidad constante
    cinta.setAcceleration(50) # opcional, mm/s^2
    cinta.MoveJ(cinta.Joints() + INCREMENTO_MM)

--- Python program ResetPick ---
# Type help("robodk.robolink") or help("robodk.robomath") for more information
# Press F5 to run the script
# Documentation: https://robodk.com/doc/en/RoboDK-API.html
# Reference:     https://robodk.com/doc/en/PythonAPI/robodk.html
# Note: It is not required to keep a copy of this file, your Python script is saved with your RDK project

# You can also use the new version of the API:
from robodk import robolink    # RoboDK API
from robodk import robomath    # Robot toolbox
RDK = robolink.Robolink()

cinta = RDK.Item('cinta 2')

if cinta.Valid():
    cinta.setJoints([2000])

--- Python program AvanzaPick ---
# Type help("robodk.robolink") or help("robodk.robomath") for more information
# Press F5 to run the script
# Documentation: https://robodk.com/doc/en/RoboDK-API.html
# Reference:     https://robodk.com/doc/en/PythonAPI/robodk.html
# Note: It is not required to keep a copy of this file, your Python script is saved with your RDK project

# You can also use the new version of the API:
from robodk import robolink    # RoboDK API
from robodk import robomath    # Robot toolbox
RDK = robolink.Robolink()

cinta = RDK.Item('cinta 2')
INCREMENTO_MM = -70
#caja = RDK.Item('Frame 11')
SR_Cinta = RDK.Item('Frame 11')

if cinta.Valid():
    cinta.setSpeed(500)        # velocidad constante
    cinta.setAcceleration(500) # opcional, mm/s^2
    cinta.MoveJ(cinta.Joints() + INCREMENTO_MM)

--- Python program ProgramaClasificacion ---
from robodk import *
from robolink import *

RDK = Robolink()
robot = RDK.Item('UR3e Base - Clasificación', ITEM_TYPE_ROBOT)

tool = RDK.Item("RobotiQ EPick Vacuum Gripper (1 Cup)", ITEM_TYPE_TOOL)
frame_est = RDK.Item('Sistema - Estantería')

#base = RDK.Item('Estanteria')
#pose_base = base.Pose()


#pose_base = pose_base * transl(0, 0, 280)

#♥ TARGETS

target_Punto_Paso_1 = RDK.Item('Paso', robolink.ITEM_TYPE_TARGET)
target_Punto_Paso_2 = RDK.Item('Target 2', robolink.ITEM_TYPE_TARGET)
target_Punto_Paso_3 = RDK.Item('Target 3', robolink.ITEM_TYPE_TARGET)
#target_Pre_Place = RDK.Item('PrePlace', robolink.ITEM_TYPE_TARGET)


target_Place = RDK.Item('Place_base', robolink.ITEM_TYPE_TARGET)
pose_base = target_Place.Pose()


# Parámetros
ancho_caja = 125
fondo_caja = 66
alto_caja = 62.5

gap = 30

dx = ancho_caja + gap
dy = fondo_caja + gap
dz = 215

cols = 3
rows = 2
levels = 3

contador = 0
max_cajas = 18

robot.setPoseFrame(frame_est)
robot.setPoseTool(tool)

pose_target = pose_base

for k in range(levels):
    for i in range(rows):
        for j in range(cols):

            if contador >= max_cajas:
                break

            # PICK

            if contador % 2 == 0:
                RDK.RunProgram("Pick1", True)
            else:
                RDK.RunProgram("Pick2", True)
                if contador == 5:
                    RDK.RunProgram("AvanzaPlace", True)
                    RDK.RunProgram("AvanzaPlace", True)
                    RDK.RunProgram("AvanzaPlace", False)
                elif contador == 9:
                    RDK.RunProgram("AvanzaPlace", True)
                    RDK.RunProgram("AvanzaPlace", False)
                elif(contador == 15):
                    RDK.RunProgram("AvanzaPlace", True)
                    RDK.RunProgram("AvanzaPick", False)
                else:
                    RDK.RunProgram("AvanzaPick", False)

            #tool.AttachClosest()   # o caja.AttachTo(tool)

            # -------------------
            # CALCULAR PLACE
            # -------------------
            #offset = transl(
                #j*dx + ancho_caja/2,
                #i*dy + fondo_caja/2,
                #k*dz + alto_caja/2
            #)

            if contador <= 5:
                offset = transl(
                    j*dx + ancho_caja/2,
                    -i*dz + fondo_caja,
                    0
                )
            elif contador > 5 and contador <= 11 :
                offset = transl(
                    j*dx + ancho_caja/2,
                    -i*dz,
                    0
                )
            elif contador > 11 and contador <= 17:
                if contador == 16 or contador == 17:
                    offset = transl(
                        j*dx + ancho_caja/2,
                        -i*dz - fondo_caja + 7,
                        0
                    )
                else:
                    offset = transl(
                        j*dx + ancho_caja/2,
                        -i*dz - fondo_caja,
                        0
                    )
            else:
                offset = transl(
                    j*dx + ancho_caja/2,
                    -i*dz + fondo_caja,
                    0
                )


            pose_target = pose_base * offset

            robot.setPoseFrame(frame_est)
            robot.setPoseTool(tool)

            # -------------------
            # PLACE
            # -------------------
            robot.MoveJ(target_Punto_Paso_3)

            robot.MoveJ(target_Punto_Paso_2)
            robot.MoveJ(pose_target * robomath.transl([0,-50,0]))
            robot.setSpeed(100,20)
            pause(0.5)
            robot.MoveL(pose_target)

            objetos = tool.Childs()
            if len(objetos) > 0:
                caja = objetos[0]
                caja.setParentStatic(frame_est)

            tool.DetachAll()

            robot.MoveL(pose_target * robomath.transl([0,-50,0]))
            robot.setSpeed(1000,100)
            robot.MoveJ(target_Punto_Paso_2)

            # o mejor:
            # caja.AttachTo(frame_est)

            contador += 1

--- Python program Pedidos_PickPlace_base ---
from robodk import *
from robolink import *

RDK = Robolink()

robot = RDK.Item('UR3e - pedidos', ITEM_TYPE_ROBOT)
tool = robot.getLink(ITEM_TYPE_TOOL)
frame_est = RDK.Item('Sistema - Estantería')
frame_pedidos = RDK.Item('Frame_pedidos')

t_paso3 = RDK.Item('Paso_ped3', ITEM_TYPE_TARGET)
t_paso4 = RDK.Item('Paso_ped4', ITEM_TYPE_TARGET)
t_paso5 = RDK.Item('Paso_ped5', ITEM_TYPE_TARGET)
t_paso6 = RDK.Item('Paso_ped6', ITEM_TYPE_TARGET)

t_reposo  = RDK.Item('Reposo_pedidos', ITEM_TYPE_TARGET)
t_paso1   = RDK.Item('Paso_ped1', ITEM_TYPE_TARGET)
t_paso2   = RDK.Item('Paso_ped2', ITEM_TYPE_TARGET)
t_preplace = RDK.Item('Pre_pedidos', ITEM_TYPE_TARGET)
t_place = RDK.Item('Place_pedido', ITEM_TYPE_TARGET)

t_pick_ref = RDK.Item('Pick_base_antes', ITEM_TYPE_TARGET)
pose_ref = t_pick_ref.Pose()

robot.setPoseFrame(frame_est)
robot.setPoseTool(tool)

pose_base = RDK.Item('Place_base', ITEM_TYPE_TARGET).Pose()
pose_target = pose_base

# BASE DE DATOS

medicamentos = {
    "ibuprofeno": [],
    "paracetamol": [],
    "enantyum": []
}


# PARÁMETROS

ancho_caja = 125
fondo_caja = 66
alto_caja = 62.5
gap = 30
dx = ancho_caja + gap
dz = 215
cols = 3
rows = 2
levels = 3
contador = 0
max_cajas = 18

# GENERAR POSICIONES

for k in range(levels):
    for i in range(rows):
        for j in range(cols):
            if contador >= max_cajas:
                break

            if contador <= 5:
                offset = transl(j*dx + ancho_caja/2, -i*dz + fondo_caja, 0)
                if contador == 0 or contador == 3:
                    medicamentos["ibuprofeno"].append(pose_target * offset)
                elif contador <= 2:
                    medicamentos["paracetamol"].append(pose_target * offset)
                else:
                    medicamentos["enantyum"].append(pose_target * offset)

            elif contador <= 11:
                offset = transl(j*dx + ancho_caja/2, -i*dz, 0)
                if contador == 6 or contador == 9:
                    medicamentos["ibuprofeno"].append(pose_target * offset)
                elif contador <= 8:
                    medicamentos["paracetamol"].append(pose_target * offset)
                else:
                    medicamentos["enantyum"].append(pose_target * offset)

            elif contador <= 17:
                if contador == 16 or contador == 17:
                    offset = transl(j*dx + ancho_caja/2, -i*dz - fondo_caja + 7, 0)
                else:
                    offset = transl(j*dx + ancho_caja/2, -i*dz - fondo_caja, 0)
                if contador == 12 or contador == 15:
                    medicamentos["ibuprofeno"].append(pose_target * offset)
                elif contador <= 14:
                    medicamentos["paracetamol"].append(pose_target * offset)
                else:
                    medicamentos["enantyum"].append(pose_target * offset)

            contador += 1

# FUNCIÓN PEDIDO

def pedir_medicamento(tipo):
    if tipo not in medicamentos or not medicamentos[tipo]:
        print("Sin stock de", tipo)
        return

    pose_place_pos = medicamentos[tipo].pop()

    pose_place = Mat(pose_ref)
    pose_place[0,3] = pose_place_pos[0,3]
    pose_place[1,3] = pose_place_pos[1,3]
    pose_place[2,3] = pose_place_pos[2,3]

    pose_up = Mat(pose_place)
    pose_up[1,3] += 100
    pose_pick = Mat(pose_place)
    pose_pick[1,3] += 60

    robot.MoveJ(t_paso3)
    robot.MoveJ(t_paso4)
    robot.MoveJ(t_paso5)
    robot.MoveJ(t_paso6)

    robot.MoveJ(pose_up)
    robot.setSpeed(100, 20)
    pause(0.5)
    robot.MoveL(pose_pick)

    tool.AttachClosest()
    robot.MoveL(pose_up)
    robot.setSpeed(1000, 100)

    robot.MoveJ(t_paso6)
    robot.MoveJ(t_paso5)
    robot.MoveJ(t_paso4)
    robot.MoveJ(t_paso3)

    robot.setPoseFrame(frame_pedidos)

    # PLACE
    robot.MoveJ(t_reposo)
    robot.MoveJ(t_paso1)
    robot.MoveJ(t_paso2)

    robot.MoveJ(t_preplace)
    robot.setSpeed(100, 20)
    pause(0.5)
    robot.MoveL(t_place)

    tool.DetachAll()
    robot.MoveL(t_preplace)
    robot.setSpeed(1000, 100)

    robot.MoveJ(t_paso2)
    robot.MoveJ(t_paso1)
    robot.MoveJ(t_reposo)

#  EJECUTAR

pedir_medicamento("enantyum")

--- Python program Pedidos_PickPlace ---
from robodk import *
from robolink import *

RDK = Robolink()

robot = RDK.Item('UR3e - pedidos', ITEM_TYPE_ROBOT)
tool = robot.getLink(ITEM_TYPE_TOOL)
frame_est = RDK.Item('Sistema - Estantería')
frame_pedidos = RDK.Item('Frame_pedidos')

t_paso3 = RDK.Item('Paso_ped3', ITEM_TYPE_TARGET)
t_paso4 = RDK.Item('Paso_ped4', ITEM_TYPE_TARGET)
t_paso5 = RDK.Item('Paso_ped5', ITEM_TYPE_TARGET)
t_paso6 = RDK.Item('Paso_ped6', ITEM_TYPE_TARGET)

t_reposo  = RDK.Item('Reposo_pedidos', ITEM_TYPE_TARGET)
t_paso1   = RDK.Item('Paso_ped1', ITEM_TYPE_TARGET)
t_paso2   = RDK.Item('Paso_ped2', ITEM_TYPE_TARGET)
t_preplace = RDK.Item('Pre_pedidos', ITEM_TYPE_TARGET)
t_place = RDK.Item('Place_pedido', ITEM_TYPE_TARGET)

t_pick_ref = RDK.Item('Pick_base_antes', ITEM_TYPE_TARGET)
pose_ref = t_pick_ref.Pose()

robot.setPoseFrame(frame_est)
robot.setPoseTool(tool)

pose_base = RDK.Item('Place_base', ITEM_TYPE_TARGET).Pose()
pose_target = pose_base

# BASE DE DATOS

medicamentos = {
    "ibuprofeno": [],
    "paracetamol": [],
    "enantyum": []
}

alias_medicamentos = {
    "amoxicilina": "enantyum"
}

medicamento_por_id = {
    1: "paracetamol",
    2: "ibuprofeno",
    3: "enantyum"
}


# PARÁMETROS

ancho_caja = 125
fondo_caja = 66
alto_caja = 62.5
gap = 30
dx = ancho_caja + gap
dz = 215
cols = 3
rows = 2
levels = 3
contador = 0
max_cajas = 18

# GENERAR POSICIONES

for k in range(levels):
    for i in range(rows):
        for j in range(cols):
            if contador >= max_cajas:
                break

            if contador <= 5:
                offset = transl(j*dx + ancho_caja/2, -i*dz + fondo_caja, 0)
                if contador == 0 or contador == 3:
                    medicamentos["ibuprofeno"].append(pose_target * offset)
                elif contador <= 2:
                    medicamentos["paracetamol"].append(pose_target * offset)
                else:
                    medicamentos["enantyum"].append(pose_target * offset)

            elif contador <= 11:
                offset = transl(j*dx + ancho_caja/2, -i*dz, 0)
                if contador == 6 or contador == 9:
                    medicamentos["ibuprofeno"].append(pose_target * offset)
                elif contador <= 8:
                    medicamentos["paracetamol"].append(pose_target * offset)
                else:
                    medicamentos["enantyum"].append(pose_target * offset)

            elif contador <= 17:
                if contador == 16 or contador == 17:
                    offset = transl(j*dx + ancho_caja/2, -i*dz - fondo_caja + 7, 0)
                else:
                    offset = transl(j*dx + ancho_caja/2, -i*dz - fondo_caja, 0)
                if contador == 12 or contador == 15:
                    medicamentos["ibuprofeno"].append(pose_target * offset)
                elif contador <= 14:
                    medicamentos["paracetamol"].append(pose_target * offset)
                else:
                    medicamentos["enantyum"].append(pose_target * offset)

            contador += 1

# FUNCIÓN PEDIDO

def pedir_medicamento(tipo):
    tipo = alias_medicamentos.get(tipo, tipo)

    if tipo not in medicamentos or not medicamentos[tipo]:
        print("Sin stock de", tipo)
        RDK.setParam("pedido_resultado", "sin_stock")
        return False

    pose_place_pos = medicamentos[tipo].pop()

    pose_place = Mat(pose_ref)
    pose_place[0,3] = pose_place_pos[0,3]
    pose_place[1,3] = pose_place_pos[1,3]
    pose_place[2,3] = pose_place_pos[2,3]

    pose_up = Mat(pose_place)
    pose_up[1,3] += 100
    pose_pick = Mat(pose_place)
    pose_pick[1,3] += 60

    robot.MoveJ(t_paso3)
    robot.MoveJ(t_paso4)
    robot.MoveJ(t_paso5)
    robot.MoveJ(t_paso6)

    robot.MoveJ(pose_up)
    robot.setSpeed(100, 20)
    pause(0.5)
    robot.MoveL(pose_pick)

    tool.AttachClosest()
    robot.MoveL(pose_up)
    robot.setSpeed(1000, 100)

    robot.MoveJ(t_paso6)
    robot.MoveJ(t_paso5)
    robot.MoveJ(t_paso4)
    robot.MoveJ(t_paso3)

    robot.setPoseFrame(frame_pedidos)

    # PLACE
    robot.MoveJ(t_reposo)
    robot.MoveJ(t_paso1)
    robot.MoveJ(t_paso2)

    robot.MoveJ(t_preplace)
    robot.setSpeed(100, 20)
    pause(0.5)
    robot.MoveL(t_place)

    tool.DetachAll()
    robot.MoveL(t_preplace)
    robot.setSpeed(1000, 100)

    robot.MoveJ(t_paso2)
    robot.MoveJ(t_paso1)
    robot.MoveJ(t_reposo)
    RDK.setParam("pedido_resultado", "ok")
    return True

def tipo_desde_parametros():
    pedido_id = RDK.getParam("pedido_id")
    try:
        pedido_id = int(str(pedido_id).strip())
    except (TypeError, ValueError):
        pedido_id = 0

    if pedido_id in medicamento_por_id:
        return medicamento_por_id[pedido_id], pedido_id

    tipo = RDK.getParam("pedido_tipo")
    if tipo is None or tipo == "":
        return "enantyum", 3

    tipo = str(tipo).strip().lower()
    return alias_medicamentos.get(tipo, tipo), 0


#  EJECUTAR

tipo_recibido, id_recibido = tipo_desde_parametros()
print("Medicamento recibido:", tipo_recibido, "id:", id_recibido)

pedir_medicamento(tipo_recibido)

--- program ProgramaPrincipal (robot UR3e - Clasificaci) ---
  Llamar Programa Despaletizado
  Llamar ProgramaClasificacion
